// TIA Portal V17 export
// export: Created 2025-06-26T06:49:33.2156309Z, ExportSetting WithDefaults, DisplayName Totally Integrated Automation Portal, DisplayVersion V17 Update 8, DisplayName TIA Portal Openness, DisplayVersion V17 Update 8, DisplayName TIA Portal Version Control Interface, DisplayVersion V17, DisplayName STEP 7 Professional, DisplayVersion V17 Update 8, DisplayName STEP 7 Safety, DisplayVersion V17 Update 6, DisplayName WinCC Advanced, DisplayVersion V17 Update 8
VAR_GLOBAL   // PLC tag table "Customer"
   "VB3-M8301 Start" AT %I200.0 : Bool;   // Anfrage starten 1 = Wärmepumpe starten, 0 = nichts tun
   "VB3-M8301 Stop" AT %I200.1 : Bool;   // Stopp-Anfrage 1 = stoppen, 0 = nichts tun (überschreibt das Startsignal)
   "VB3-M8301 Freigabe" AT %I200.2 : Bool;   // Freigabe 1 = Startbefehl aktivieren 0 = Startbefehl ignorieren
   "VB3-M8301 Reset" AT %I200.3 : Bool;   // Alarmbestätigung 1 = alle Alarme löschen, 0 = nichts tun
   "VB3-M8301 Not-Aus" AT %I200.4 : Bool;   // Not-Aus zurücksetzen 1 = Not-Aus zurücksetzen, 0 = nichts tun
   "VB3-M8301 Sstop" AT %I200.5 : Bool;   // Schnellstopp-Anfrage 1 = Schnellstoppanforderung, 0 = nichts tun
   "A1024.6" AT %I200.6 : Bool;   // Reserve
   "A1024.7" AT %I200.7 : Bool;   // Reserve
   QI117_828B2 AT %I203.0 : Bool;   // Rückmeldung zur Raumlüftung WP1 1 = Lüftung ok, 0 = Startbefehl ignorieren
   QI117_828B3 AT %I203.1 : Bool;   // Kondensierbare Gase erkannt WP1 1 = Anforderung stoppen und Absperrventile schließen, 0 = nichts tun
   "A1027.2" AT %I203.2 : Bool;   // Reserve
   "A1027.3" AT %I203.3 : Bool;   // Reserve
   "A1027.4" AT %I203.4 : Bool;   // Reserve
   "A1027.5" AT %I203.5 : Bool;   // Reserve
   "A1027.6" AT %I203.6 : Bool;   // Reserve
   "VB3-M8301 Live bit" AT %I203.7 : Bool;   // Live bit
   QI117_828B1 AT %IW201 : Int;   // [%] Leistungssollwert WP1 Sollwert für die Systemleistung
   AW1028 AT %IW204 : Int;   // Reserve
   AW1030 AT %IW206 : Int;   // Reserve
   "VB3-M8301 NA-Status" AT %Q200.0 : Bool;   // Not-Aus-Status 1 = Not-Aus ok, 0 = Not-Aus aktiv
   "VB3-M8301 G1 Ein" AT %Q200.1 : Bool;   // Status der Ölheizungen Gruppe 1 1 = Heizungen ein, 0 = Heizungen aus
   "VB3-M8301 G2 Ein" AT %Q200.2 : Bool;   // Status der Ölheizungen Gruppe 2 1 = Heizungen ein, 0 = Heizungen aus
   "E1024.3" AT %Q200.3 : Bool;   // Reserve
   "E1024.4" AT %Q200.4 : Bool;   // Reserve
   "E1024.5" AT %Q200.5 : Bool;   // Reserve
   "E1024.6" AT %Q200.6 : Bool;   // Reserve
   "E1024.7" AT %Q200.7 : Bool;   // Reserve
   GH117_827 AT %Q201.0 : Bool;   // Absalzventil 1 = offen, 0 = geschlossen, gesteuert durch Heaten
   GH117_826_1 AT %Q201.1 : Bool;   // Ventil nicht kondensierbares Gase 1 1 = offen, 0 = geschlossen, gesteuert durch Heaten
   GH117_826_2 AT %Q201.2 : Bool;   // Ventil nicht kondensierbares Gase 2 1 = offen, 0 = geschlossen, gesteuert durch Heaten
   "E1025.3" AT %Q201.3 : Bool;   // Reserve
   "E1025.4" AT %Q201.4 : Bool;   // Reserve
   "E1025.5" AT %Q201.5 : Bool;   // Reserve
   "E1025.6" AT %Q201.6 : Bool;   // Reserve
   "E1025.7 Live Bit" AT %Q201.7 : Bool;   // Live bit
   "VB3-M8301 Status" AT %QW202 : Int;   // Maschinenzustand 0 = Initialisierung, 1 = Offline, 2 = Standby, Aufwärmen, Betrieb usw. (Aufzählungstyp)
   QI117_828B4 AT %QW204 : Int;   // [h] Betriebsstunden Zählt, solange der Heatbooster eingeschaltet ist
   QI117_828B5 AT %QW206 : Int;   // [h] Aktive Zeit Stunden Aktiv bedeutet, dass die Maschine eingeschaltet ist (entweder im Betrieb oder im Leerlauf).
   QI117_828B6 AT %QW208 : Int;   // [h] Laufzeit Stunden Laufen bedeutet in Betrieb (Wärmeerhöhung!)
   QI117_828B7 AT %QW210 : Int;   // [C] HBL-TT-07 (HBL-TT-901) Temperatur Saugseite Kondensator
   QI117_828B8 AT %QW212 : Int;   // [C] HBL-TT-08 (HBL-TT-518) Temperatur Druckseit Kondensator
   QI117_828B9 AT %QW214 : Int;   // [C] HBL-TT-13 (HBL-TT-546) Temperatur Saugseite Verdampfer
   QI117_828B10 AT %QW216 : Int;   // [C] HBL-TT-14 (HBL-TT-542) Temperatur Druckseit Verdampfer
   QI117_828B11 AT %QW218 : Int;   // [C] HBL-TT-16 Lufttemperatur des Containers
   QI117_828B12 AT %QW220 : Int;   // [C] HBL-TT-17 Lufttemperatur im Schaltschrank
   QI117_828B13 AT %QW222 : Int;   // [C] HBL-TT-18 Umgebungslufttemperatur
   QI117_828B16 AT %QW224 : Int;   // [ppm] HBL-CT-03 Gasdetektor Container
   QI117_828B17 AT %QW226 : Int;   // [%] SSC-LT-01 Füllstand des Sperrflüssigkeitsbehälters
   "VB3-M8301 Wärme" AT %QW228 : Int;   // [kW] Voraussichtliche Wärmelieferung
   QI117_828B18 AT %QW230 : Int;   // [1] System: COP
   "VB3-M8301 kW" AT %QW232 : Int;   // [kW] System: electrical power
   QI117_828B19 AT %QW234 : Int;   // [C] System: temperature lift
   GH117_812 AT %QW236 : Int;   // [%] Kondensatventil Verdampfer ein
   GH117_818 AT %QW238 : Int;   // [%] Dampfventil Verdampfer aus (HBL-HCV-514)
   GH117_815 AT %QW240 : Int;   // [%] Dampfventil Kondensator ein (HBL-HCV-548)
   GH117_821 AT %QW242 : Int;   // [%] Kondensatventil Kondensator aus
   EW1072 AT %QW248 : Int;   // Reserve
   "VB3-M8301 kW(1)" AT %QW244 : Int;   // Elektrische Leistung
   EW1070 AT %QW246 : Int;   // Reserve
   EW1074 AT %QW250 : Int;   // Reserve
END_VAR
